# EPICS substitutions: ek9000App/Db/EL3114.substitutions
file EL3114.template
{       pattern
        {
                TERMINAL,

        }
        {
        }
}
